{attribute 'GeneratedUsingTerminal: EK1100-0000-0018'}
{attribute addProperty BoxType "EK1100-0000-0018"}
{attribute addProperty Id "RC50_A2_EK1122RC50_A2_EK1122_AE8686CC73RC50_A3_EK1122RC50_A3_EK1122_7F1D927D120RC50_A5_EL1809EL1809_32157CFD20RC50_A6_EL1809EL1809_32157CFD20RC50_A7_EL2809EL2809_2B6483BD19RC50_A8_EL2809EL2809_2B6483BD19RC50_A9_EL2809EL2809_2B6483BD19RC50_1_EndTerminal_EL9010EL9010_D29C20850"}
{attribute addProperty CRC "3605416262"}
{attribute addProperty Size "290"}
{attribute addProperty Name "RC50_1 (EK1100)"}
TYPE RC50_1_EK1100_D6E64946 EXTENDS EK1100_1FC0878B : 
STRUCT
    {attribute addProperty Name "RC50_A2 (EK1122)"}
    {attribute addProperty PreviousPort "RC50_1 (EK1100) : B"}
    {attribute addProperty SyncUnit "default"}
    RC50_A2_EK1122 : RC50_A2_EK1122_AE8686CC;
    {attribute addProperty Name "RC50_A3 (EK1122)"}
    {attribute addProperty PreviousPort "RC50_A2 (EK1122) : C"}
    {attribute addProperty SyncUnit "default"}
    RC50_A3_EK1122 : RC50_A3_EK1122_7F1D927D;
    {attribute addProperty Name "RC50_A5 (EL1809)"}
    {attribute addProperty PreviousPort "RC50_A3 (EK1122) : C"}
    {attribute addProperty SyncUnit "C50"}
    RC50_A5_EL1809 : EL1809_32157CFD;
    {attribute addProperty Name "RC50_A6 (EL1809)"}
    {attribute addProperty PreviousPort "RC50_A5 (EL1809) : B"}
    {attribute addProperty SyncUnit "C50"}
    RC50_A6_EL1809 : EL1809_32157CFD;
    {attribute addProperty Name "RC50_A7 (EL2809)"}
    {attribute addProperty PreviousPort "RC50_A6 (EL1809) : B"}
    {attribute addProperty SyncUnit "C50"}
    RC50_A7_EL2809 : EL2809_2B6483BD;
    {attribute addProperty Name "RC50_A8 (EL2809)"}
    {attribute addProperty PreviousPort "RC50_A7 (EL2809) : B"}
    {attribute addProperty SyncUnit "C50"}
    RC50_A8_EL2809 : EL2809_2B6483BD;
    {attribute addProperty Name "RC50_A9 (EL2809)"}
    {attribute addProperty PreviousPort "RC50_A8 (EL2809) : B"}
    {attribute addProperty SyncUnit "C50"}
    RC50_A9_EL2809 : EL2809_2B6483BD;
    {attribute addProperty Name "RC50_1_EndTerminal (EL9010)"}
    {attribute addProperty PreviousPort "RC50_A9 (EL2809) : B"}
    {attribute addProperty SyncUnit "default"}
    RC50_1_EndTerminal_EL9010 : EL9010_D29C2085;
END_STRUCT
END_TYPE

(* stored: Version 1.2.0.0, ProductVersion 3.1.4024.11
   DUT RC50_1_EK1100_D6E64946: Id {c2a47b8f-c5e7-0b34-26f6-0e98bfc38a74} *)
